PROGRAM Conveyor_1
VAR
	Always_ON	:	BOOL	:=TRUE	;//상시 ON 
	Always_OFF	:	BOOL	:=FALSE	;//상시 OFF
END_VAR

// NETWORK 1

// NETWORK 2

// NETWORK 3

// NETWORK 4

// NETWORK 5

// NETWORK 6

// NETWORK 7

END_PROGRAM

(* stored: Version 1.1.0.1, ProductVersion 3.1.4024.15
   POU Conveyor_1: Id {e729a740-a522-4a4a-a0a2-cf00dc8dfbe0}, SpecialFunc None *)
